Staubli VAL3: fetchStatus.pgx

public program fetchStatus()
begin
    // fetch robot status data

    // drives_powered
    if (isPowered() == true)
      rosStatusMsg.robotStatus.nDrivesPowered = 1
    else
      rosStatusMsg.robotStatus.nDrivesPowered = 0
    endIf

    // e-stopped
    if (esStatus() == 2)
      rosStatusMsg.robotStatus.nEStopped = 1
    else
      rosStatusMsg.robotStatus.nEStopped = 0
    endIf

    // error_code
    rosStatusMsg.robotStatus.nErrorCode = -1

    // in_error
    rosStatusMsg.robotStatus.nInError = -1

    // in_motion
    if (isSettled() == true)
      rosStatusMsg.robotStatus.nInMotion = 0
    else
      rosStatusMsg.robotStatus.nInMotion = 1
    endIf

    // mode (controller/pendant mode)
    if (workingMode() == 1 or workingMode() == 2)
      rosStatusMsg.robotStatus.nMode = 1
    elseIf (workingMode() == 3 or workingMode() == 4)
      rosStatusMsg.robotStatus.nMode = 0
    else
      rosStatusMsg.robotStatus.nMode = -1
    endIf

    // motion_possible
    rosStatusMsg.robotStatus.nMotionPossible = -1
end
